FUNCTION_BLOCK Test_TExecutionWhenReady_Start_SelectsStarting EXTENDS TUnitTestbase
VAR
    Execution : TExecution;
END_VAR

// Setup...
Execution.FB_init(
    bInitRetains := FALSE,
    bInCopyCode  := FALSE);

// Test...
Execution.Start();

Assertion.AssertEquals_BOOL(
    Expected := TRUE,
    Actual   := Execution.Starting,
    VariableName  := 'Execution.Starting');

TestFinished();

END_FUNCTION_BLOCK

(* stored: Version 1.1.0.1, ProductVersion 3.1.4024.4
   POU Test_TExecutionWhenReady_Start_SelectsStarting: Id {46b1d77a-f5b0-4500-a6b6-fd7c89ce3485}, SpecialFunc None *)
